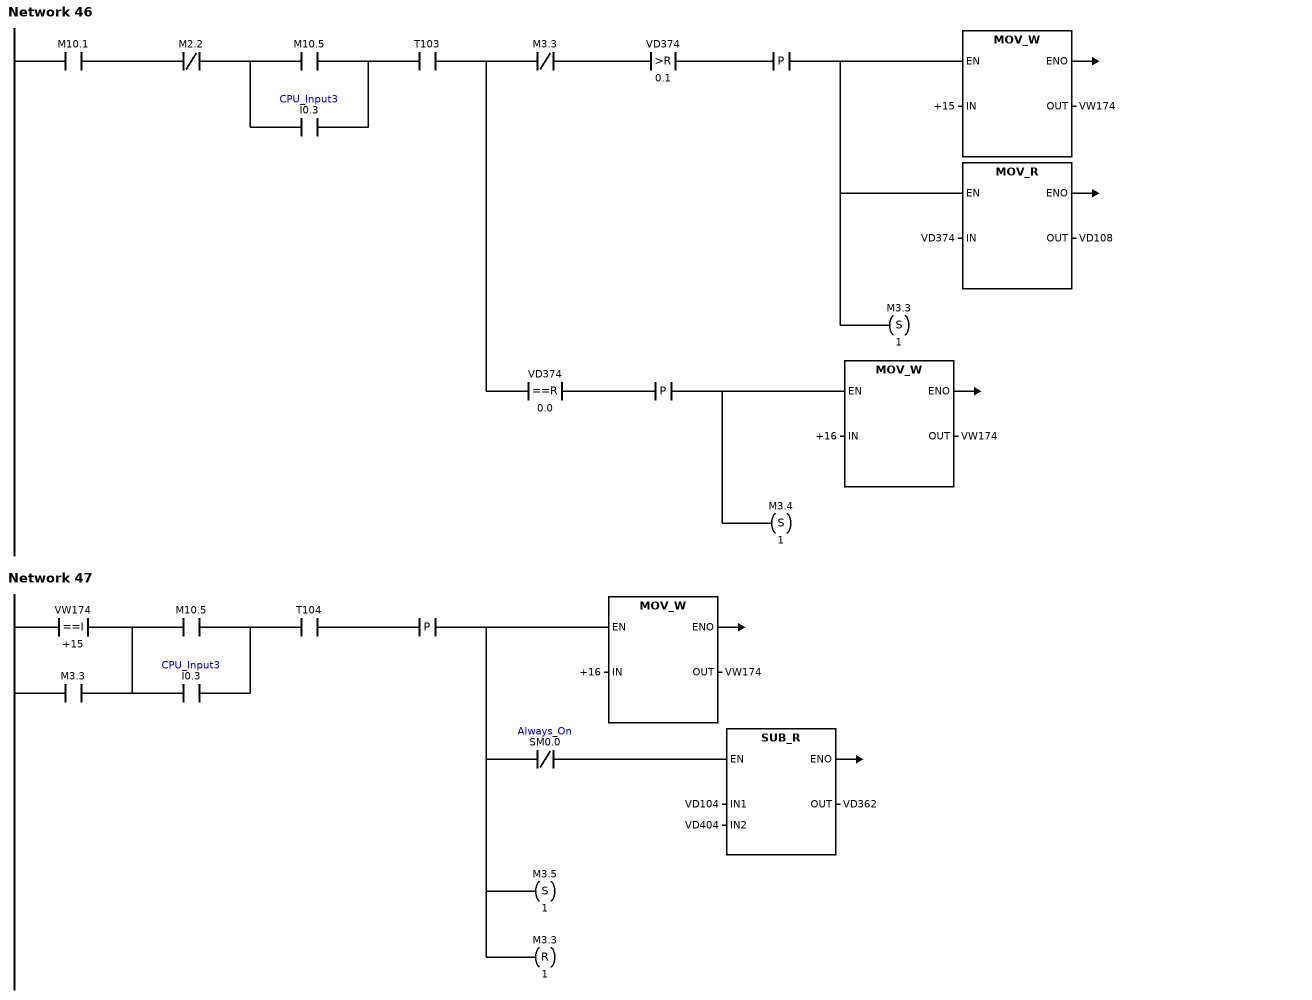
[picture p24: SBR0 networks 46-47]
Network 46
LD     M10.1
AN     M2.2
LD     M10.5
O      CPU_Input3:I0.3
ALD
A      T103
LPS
AN     M3.3
AR>    VD374, 0.1
EU
MOVW   +15, VW174
MOVR   VD374, VD108
S      M3.3, 1
LPP
AR=    VD374, 0.0
EU
MOVW   +16, VW174
S      M3.4, 1
Network 47
LDW=   VW174, +15
O      M3.3
LD     M10.5
O      CPU_Input3:I0.3
ALD
A      T104
EU
LPS
MOVW   +16, VW174
AN     Always_On:SM0.0
MOVR   VD104, VD362
-R     VD404, VD362
LRD
S      M3.5, 1
LPP
R      M3.3, 1
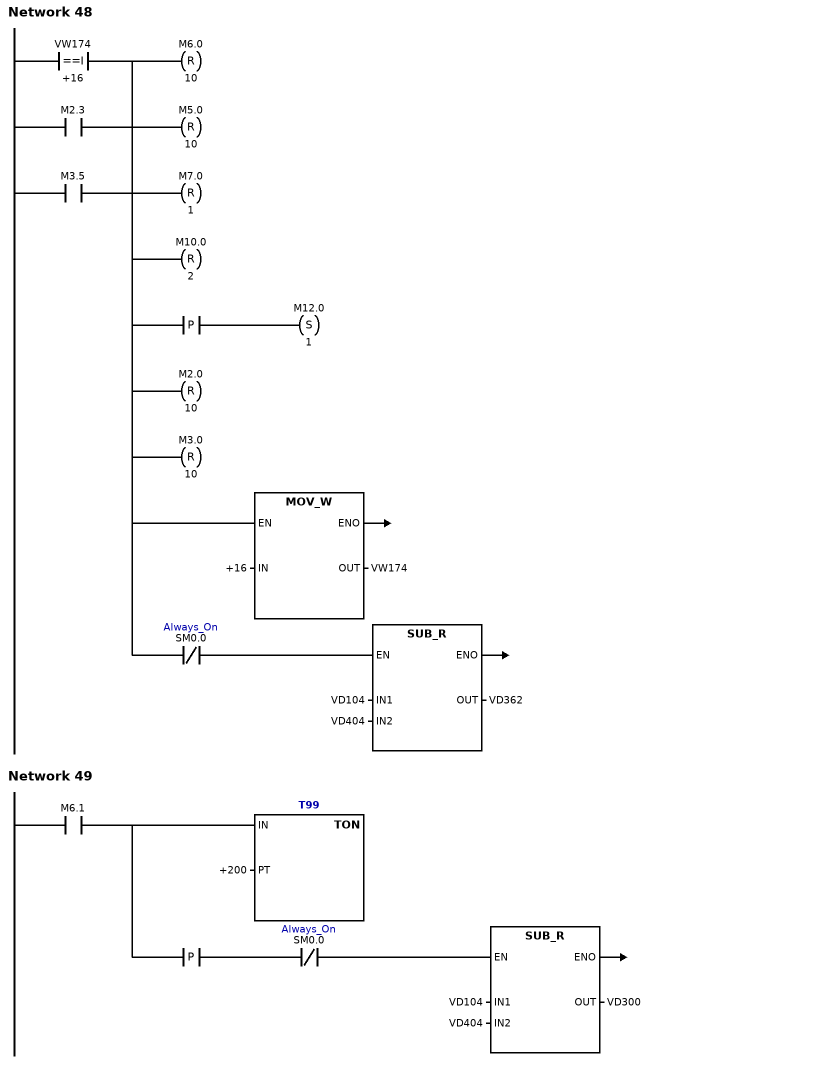
Network 48
LDW=   VW174, +16
O      M2.3
O      M3.5
LPS
R      M6.0, 10
R      M5.0, 10
R      M7.0, 1
R      M10.0, 2
EU
S      M12.0, 1
LRD
R      M2.0, 10
LRD
R      M3.0, 10
LRD
MOVW   +16, VW174
LPP
AN     Always_On:SM0.0
MOVR   VD104, VD362
-R     VD404, VD362
Network 49
LD     M6.1
TON    T99, +200
EU
AN     Always_On:SM0.0
MOVR   VD104, VD300
-R     VD404, VD300
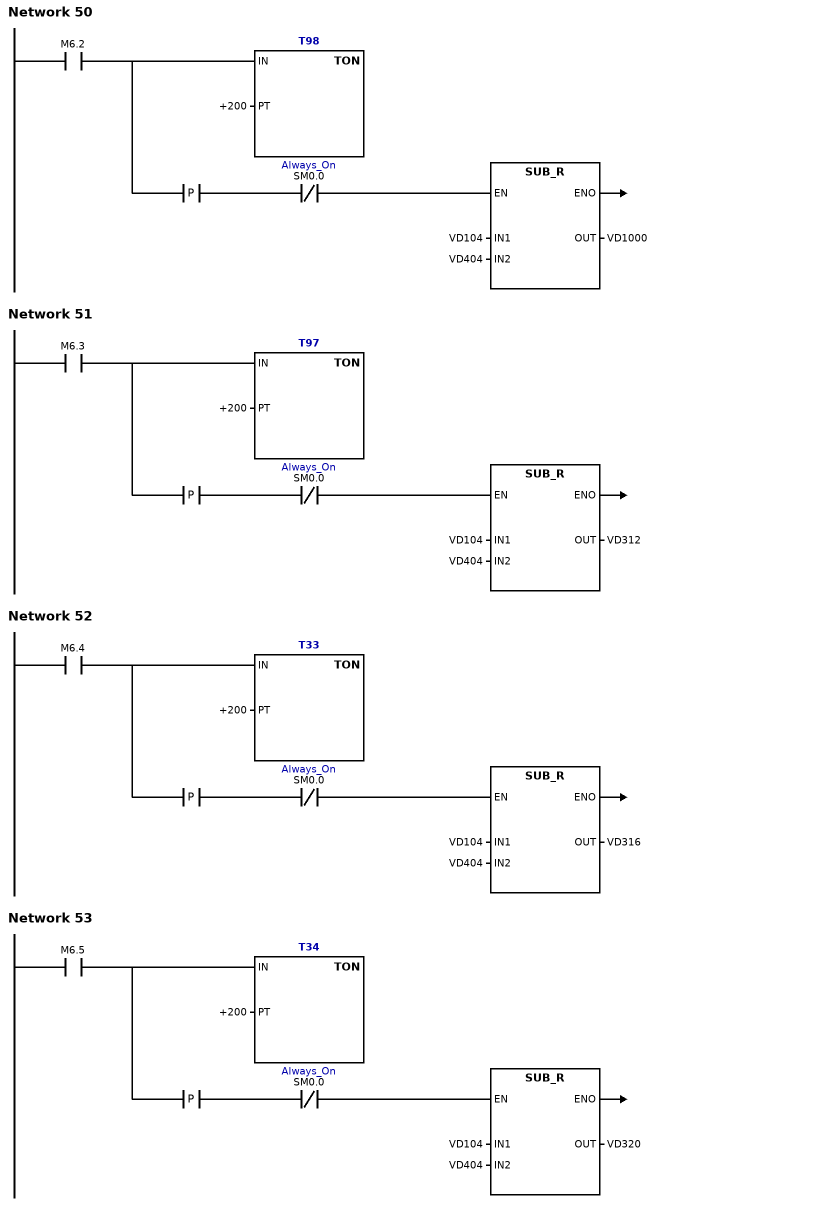
Network 50
LD     M6.2
TON    T98, +200
EU
AN     Always_On:SM0.0
MOVR   VD104, VD1000
-R     VD404, VD1000
Network 51
LD     M6.3
TON    T97, +200
EU
AN     Always_On:SM0.0
MOVR   VD104, VD312
-R     VD404, VD312
Network 52
LD     M6.4
TON    T33, +200
EU
AN     Always_On:SM0.0
MOVR   VD104, VD316
-R     VD404, VD316
Network 53
LD     M6.5
TON    T34, +200
EU
AN     Always_On:SM0.0
MOVR   VD104, VD320
-R     VD404, VD320
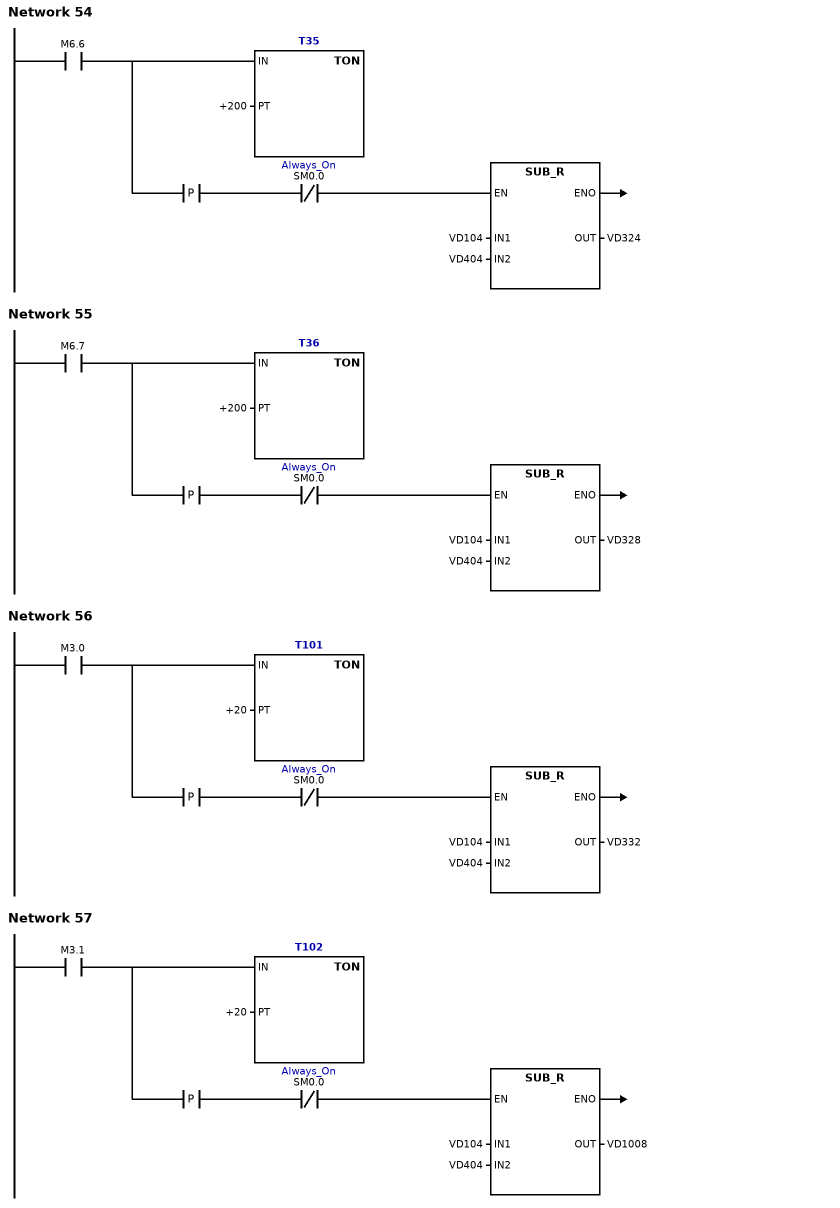
Network 54
LD     M6.6
TON    T35, +200
EU
AN     Always_On:SM0.0
MOVR   VD104, VD324
-R     VD404, VD324
Network 55
LD     M6.7
TON    T36, +200
EU
AN     Always_On:SM0.0
MOVR   VD104, VD328
-R     VD404, VD328
Network 56
LD     M3.0
TON    T101, +20
EU
AN     Always_On:SM0.0
MOVR   VD104, VD332
-R     VD404, VD332
Network 57
LD     M3.1
TON    T102, +20
EU
AN     Always_On:SM0.0
MOVR   VD104, VD1008
-R     VD404, VD1008
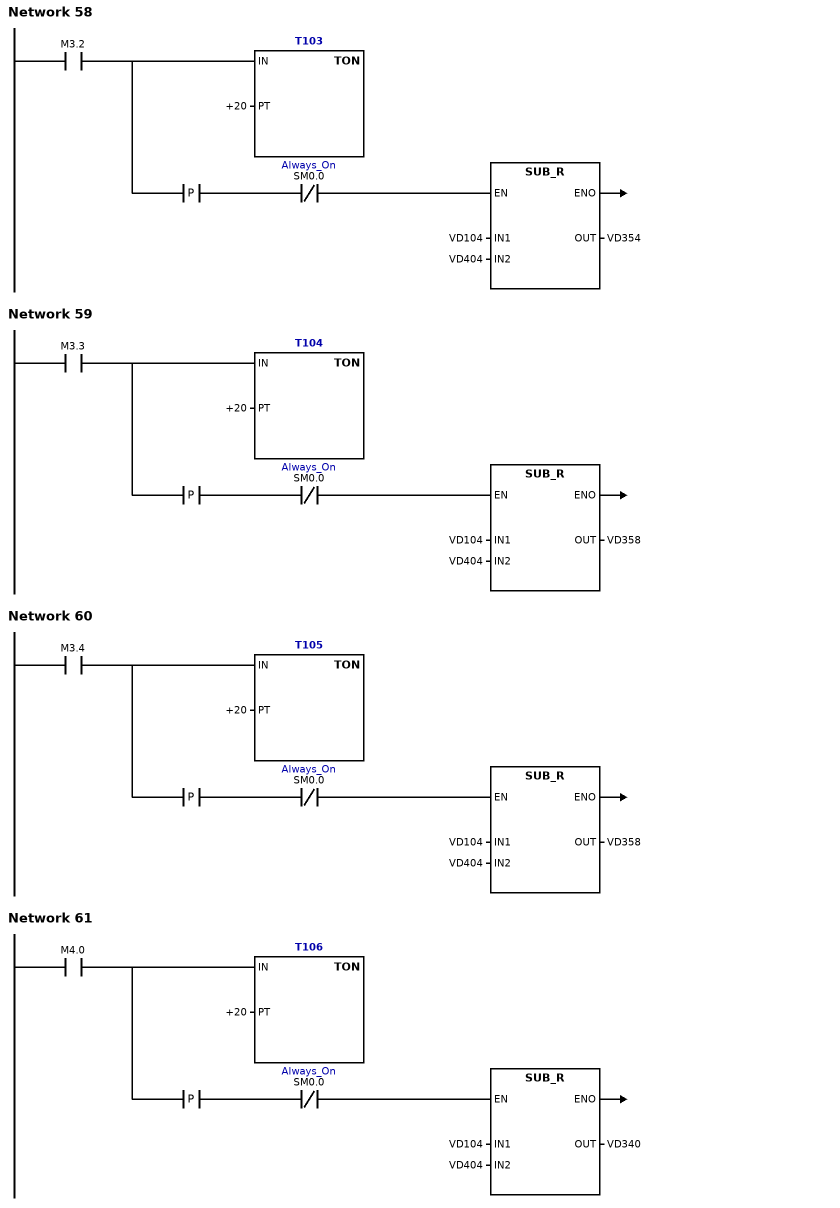
Network 58
LD     M3.2
TON    T103, +20
EU
AN     Always_On:SM0.0
MOVR   VD104, VD354
-R     VD404, VD354
Network 59
LD     M3.3
TON    T104, +20
EU
AN     Always_On:SM0.0
MOVR   VD104, VD358
-R     VD404, VD358
Network 60
LD     M3.4
TON    T105, +20
EU
AN     Always_On:SM0.0
MOVR   VD104, VD358
-R     VD404, VD358
Network 61
LD     M4.0
TON    T106, +20
EU
AN     Always_On:SM0.0
MOVR   VD104, VD340
-R     VD404, VD340
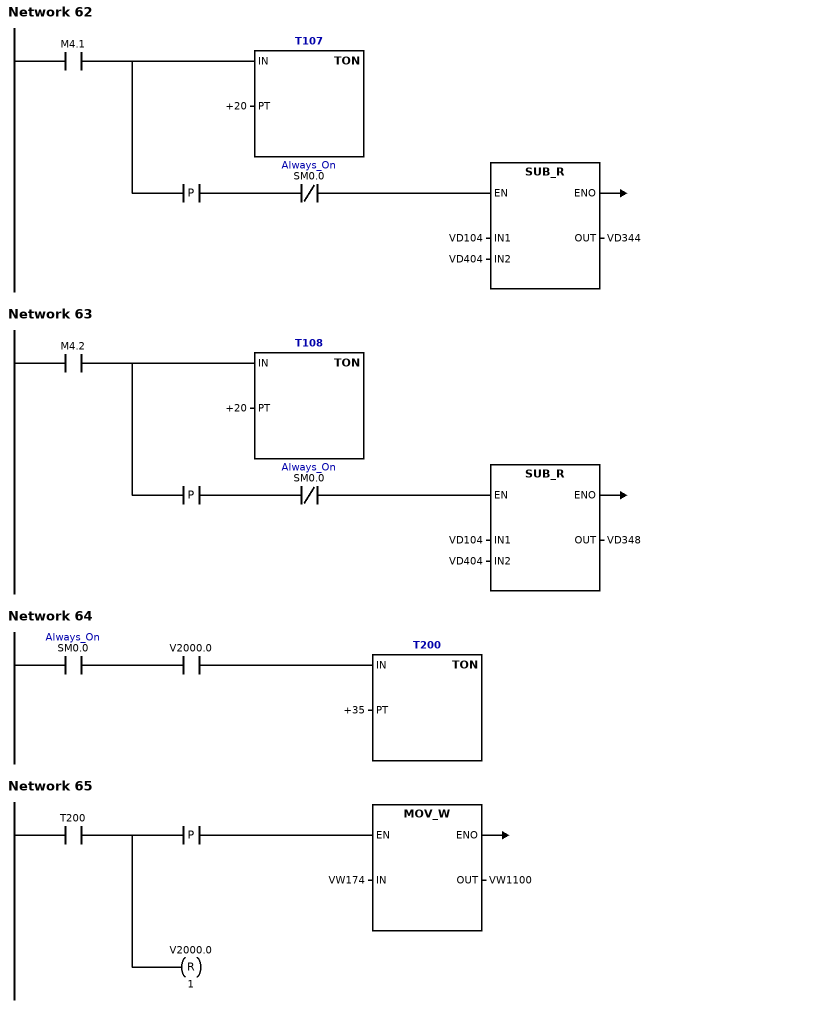
Network 62
LD     M4.1
TON    T107, +20
EU
AN     Always_On:SM0.0
MOVR   VD104, VD344
-R     VD404, VD344
Network 63
LD     M4.2
TON    T108, +20
EU
AN     Always_On:SM0.0
MOVR   VD104, VD348
-R     VD404, VD348
Network 64
LD     Always_On:SM0.0
A      V2000.0
TON    T200, +35
Network 65
LD     T200
LPS
EU
MOVW   VW174, VW1100
LPP
R      V2000.0, 1
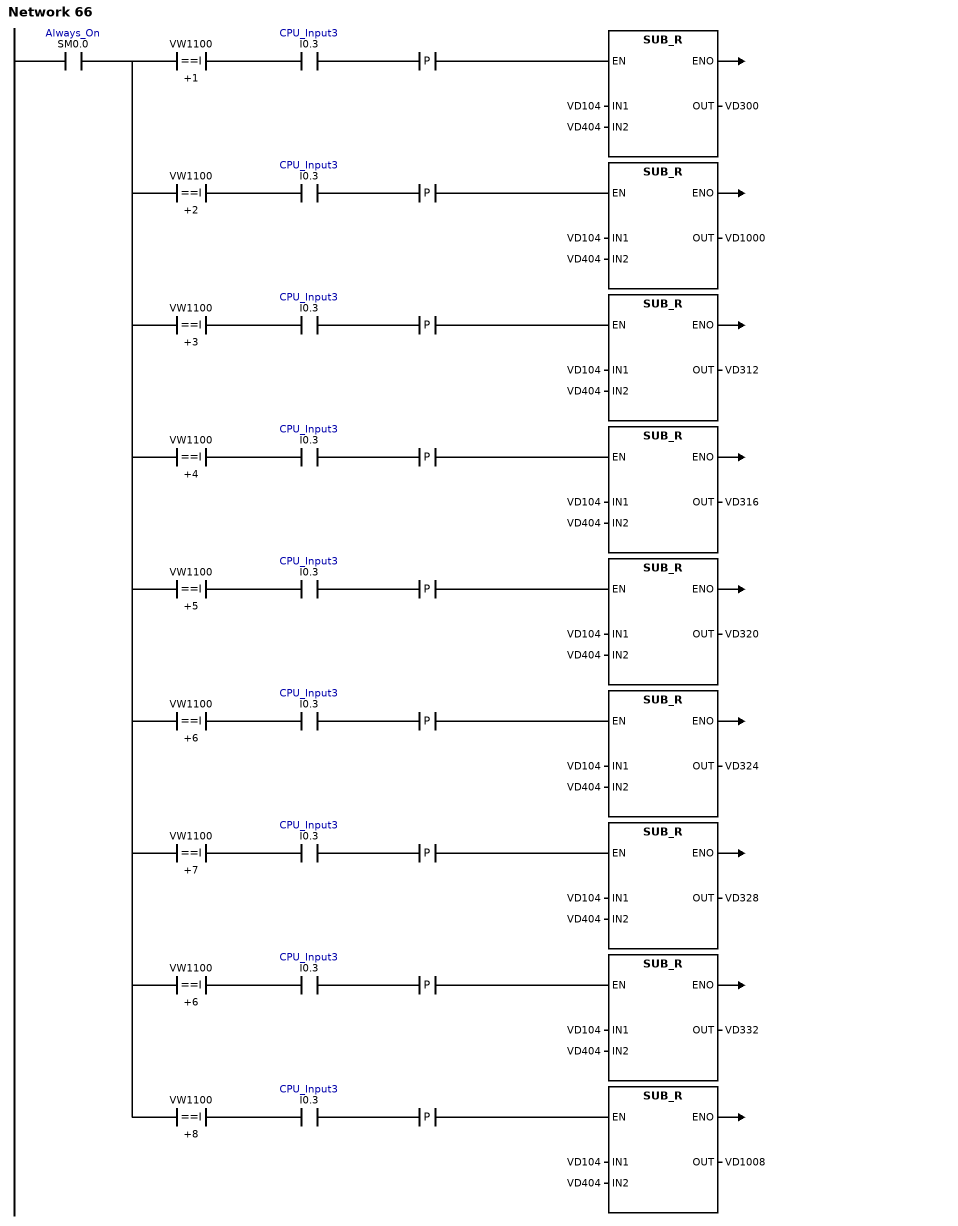
Network 66
LD     Always_On:SM0.0
LPS
AW=    VW1100, +1
A      CPU_Input3:I0.3
EU
MOVR   VD104, VD300
-R     VD404, VD300
LRD
AW=    VW1100, +2
A      CPU_Input3:I0.3
EU
MOVR   VD104, VD1000
-R     VD404, VD1000
LRD
AW=    VW1100, +3
A      CPU_Input3:I0.3
EU
MOVR   VD104, VD312
-R     VD404, VD312
LRD
AW=    VW1100, +4
A      CPU_Input3:I0.3
EU
MOVR   VD104, VD316
-R     VD404, VD316
LRD
AW=    VW1100, +5
A      CPU_Input3:I0.3
EU
MOVR   VD104, VD320
-R     VD404, VD320
LRD
AW=    VW1100, +6
A      CPU_Input3:I0.3
EU
MOVR   VD104, VD324
-R     VD404, VD324
LRD
AW=    VW1100, +7
A      CPU_Input3:I0.3
EU
MOVR   VD104, VD328
-R     VD404, VD328
LRD
AW=    VW1100, +6
A      CPU_Input3:I0.3
EU
MOVR   VD104, VD332
-R     VD404, VD332
LPP
AW=    VW1100, +8
A      CPU_Input3:I0.3
EU
MOVR   VD104, VD1008
-R     VD404, VD1008
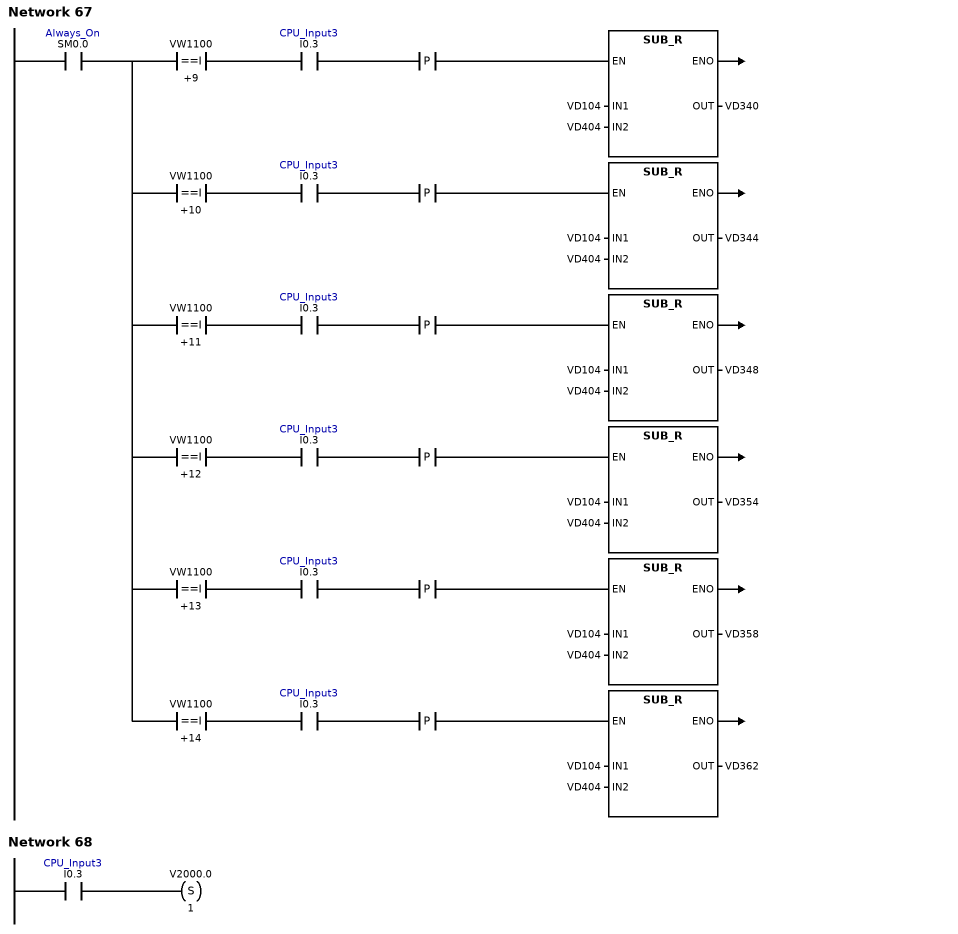
Network 67
LD     Always_On:SM0.0
LPS
AW=    VW1100, +9
A      CPU_Input3:I0.3
EU
MOVR   VD104, VD340
-R     VD404, VD340
LRD
AW=    VW1100, +10
A      CPU_Input3:I0.3
EU
MOVR   VD104, VD344
-R     VD404, VD344
LRD
AW=    VW1100, +11
A      CPU_Input3:I0.3
EU
MOVR   VD104, VD348
-R     VD404, VD348
LRD
AW=    VW1100, +12
A      CPU_Input3:I0.3
EU
MOVR   VD104, VD354
-R     VD404, VD354
LRD
AW=    VW1100, +13
A      CPU_Input3:I0.3
EU
MOVR   VD104, VD358
-R     VD404, VD358
LPP
AW=    VW1100, +14
A      CPU_Input3:I0.3
EU
MOVR   VD104, VD362
-R     VD404, VD362
Network 68
LD     CPU_Input3:I0.3
S      V2000.0, 1
END_SUBROUTINE_BLOCK
